Universal Robots URScript: 7-pickAndplace.script

def P7pickAndplace():
  set_standard_analog_input_domain(0, 1)
  set_standard_analog_input_domain(1, 1)
  set_tool_analog_input_domain(0, 1)
  set_tool_analog_input_domain(1, 1)
  set_analog_outputdomain(0, 0)
  set_analog_outputdomain(1, 0)
  set_tool_voltage(0)
  set_tcp(p[0.0,0.0,0.08,0.0,0.0,0.0])
  set_payload(0.0)
  set_gravity([0.0, 0.0, 9.82])
  $ 1 "BeforeStart"
  $ 2 "MoveJ"
  $ 3 "pick_wait_A"
  movej([-1.5531271138190403, -1.3840881815229658, -1.5578454710754102, -1.7949818880770891, 1.5962951183356604, 0.016572790374144625], a=1.3962634015954636, v=1.0471975511965976)
  while (True):
    $ 4 "机器人程序"
    $ 5 "MoveJ"
    $ 6 "pick_wait_A"
    movej([-1.5531271138190403, -1.3840881815229658, -1.5578454710754102, -1.7949818880770891, 1.5962951183356604, 0.016572790374144625], a=1.3962634015954636, v=1.0471975511965976)
    $ 7 "pick_up_A"
    movej([-1.55312711412655, -1.541128576413767, -2.225143029331143, -0.9706439349383862, 1.5962951183281175, 0.016572790066630108], a=1.3962634015954636, v=1.0471975511965976)
    $ 8 "MoveL"
    $ 9 "pick_A"
    movel([-1.553127114024047, -1.763079141223436, -2.3404225664544125, -0.6334138330028427, 1.5962951183306322, 0.016572790169128996], a=1.2, v=0.25)
    $ 10 "pick_up_A"
    movel([-1.55312711412655, -1.541128576413767, -2.225143029331143, -0.9706439349383862, 1.5962951183281175, 0.016572790066630108], a=1.2, v=0.25)
    $ 11 "MoveJ"
    $ 12 "pick_wait_A"
    movej([-1.5531271138190403, -1.3840881815229658, -1.5578454710754102, -1.7949818880770891, 1.5962951183356604, 0.016572790374144625], a=1.3962634015954636, v=1.0471975511965976, r=0.05)
    $ 13 "place_wait_B"
    movej([-0.713168896387387, -1.588181927954408, -1.3794161432946126, -1.742168910706595, 1.6060771732863524, 0.8568899972334394], a=1.3962634015954636, v=1.0471975511965976, r=0.05)
    $ 14 "place_up_B"
    movej([-0.7131689231808238, -1.7434282956805411, -2.01169665756829, -0.954641863832749, 1.6060771942141987, 0.8568900226286167], a=1.3962634015954636, v=1.0471975511965976)
    $ 15 "MoveL"
    $ 16 "place_B"
    movel([-0.7131689230968288, -1.92606917758705, -2.108818036058703, -0.6748796034328644, 1.6060771942139802, 0.8568900227126606], a=1.2, v=0.25)
    $ 17 "place_up_B"
    movel([-0.7131689231808238, -1.7434282956805411, -2.01169665756829, -0.954641863832749, 1.6060771942141987, 0.8568900226286167], a=1.2, v=0.25)
    $ 18 "MoveJ"
    $ 19 "place_wait_B"
    movej([-0.713168896387387, -1.588181927954408, -1.3794161432946126, -1.742168910706595, 1.6060771732863524, 0.8568899972334394], a=1.3962634015954636, v=1.0471975511965976, r=0.05)
    $ 20 "pick_wait_A"
    movej([-1.5531271138190403, -1.3840881815229658, -1.5578454710754102, -1.7949818880770891, 1.5962951183356604, 0.016572790374144625], a=1.3962634015954636, v=1.0471975511965976)
  end
end
